TYPE T_Ctrl_CmdListElement :
STRUCT
	///command implemented in controller
	intCmd: INT;
	///command is available info for UI
	bolAvailable: BOOL;
	
	// Name of command. Important for UI.
	strName: STRING;
END_STRUCT
END_TYPE

(* stored: Version 1.1.0.1, ProductVersion 3.1.0.14
   DUT T_Ctrl_CmdListElement: Id {ea008489-075a-49a0-a6de-0b7ede321d6d} *)
